PROGRAM MAIN
VAR
	fbMudpiReceiver: FB_MUDPI_RECEIVER;
END_VAR

fbMudpiReceiver();

END_PROGRAM

(* stored: Version 1.1.0.1, ProductVersion 3.1.4024.9
   POU MAIN: Id {8c7f3494-d62b-4dce-8edb-a017c884dc00}, SpecialFunc None *)
